// TwinCAT 3 PLC project Main
// ProgramVersion: 3.1.4022.4
// libraries:
//   Tc2_FTP, * (Beckhoff Automation GmbH)
//   Tc2_MC2, * (Beckhoff Automation GmbH)
//   Tc2_NCI, * (Beckhoff Automation GmbH)
//   Tc2_Standard, * (Beckhoff Automation GmbH)
//   Tc2_System, * (Beckhoff Automation GmbH)
//   Tc2_Utilities, * (Beckhoff Automation GmbH)
//   Tc3_IotBase, * (Beckhoff Automation GmbH)
//   Tc3_JsonXml, * (Beckhoff Automation GmbH)
//   Tc3_Module, * (Beckhoff Automation GmbH)
//   VisuSymbols,3.5.10.0,System
// project tree:
//   / GlobalTextList.TcGTLO, PlcTask.TcTTO (not stored), Visualization Manager.TcVMO (not stored)
//   GVLs/ COM.TcGVL, GVL.TcGVL
//   POUs/ commandExecute.TcPOU, ERROR.TcPOU, FTP.TcPOU, MAIN.TcPOU, POU_NCI.TcPOU, submqtt.TcPOU, commandDecoder.TcPOU
//   VISUs/ Basic.TcVIS (not stored), Visualization.TcVIS
// real-time tasks:
//   TASK PlcTask: cycle T#10ms, priority 20, ADS port 350
// motion (NC):
//   TASK NC-Task 1 SAF: cycle T#2ms, priority 4, ADS port 501
//   TASK NC-Task 1 SVB: cycle T#10ms, priority 8, ADS port 511
//   AXIS Axis X1 (id 1)
//     OtherSettings: AllowMotionCmdToSlave=true
//     encoder EncType=4
//       EncPara: ScaleFactorNumerator=40, ScaleFactorDenominator=12800, Inverse=true, MaxCount=#x0000ffff
//         SoftEndMinControl: Enable=true
//         SoftEndMaxControl: Enable=true, Range=275
//         Inc: RefSearchInverse=true, RefSyncInverse=false, RefMode=1, RefSoftSyncMask=#x0000ffff
//     drive DrvType=24
//       DrvPara: Inverse=true
//         Analog: VeloReferenz=400, ScaleFactorActTorque=0.1
//         TimeComp: TaskDelayCycles=1
//     controller CtrType=1
//       CtrPara: PriorControlFactor=1
//         PID: PosKp=25
//         Observer: BandWidth=20
//   AXIS Axis X2 (id 2)
//     OtherSettings: AllowMotionCmdToSlave=true
//     encoder EncType=4
//       EncPara: ScaleFactorNumerator=40, ScaleFactorDenominator=12800, Inverse=true, MaxCount=#x0000ffff
//         Inc: RefSoftSyncMask=#x0000ffff
//     drive DrvType=24
//       DrvPara: Inverse=true
//         Analog: VeloReferenz=400, ScaleFactorActTorque=0.1
//         TimeComp: TaskDelayCycles=1
//     controller CtrType=1
//       CtrPara: PriorControlFactor=1
//         PID: PosKp=25
//         Observer: BandWidth=20
//   AXIS Axis Y (id 4)
//     OtherSettings: AllowMotionCmdToSlave=true
//     encoder EncType=4
//       EncPara: ScaleFactorNumerator=40, ScaleFactorDenominator=12800, Inverse=true, MaxCount=#x0000ffff
//         SoftEndMinControl: Enable=true
//         SoftEndMaxControl: Enable=true, Range=275
//         Inc: RefSearchInverse=true, RefSyncInverse=false, RefMode=1, RefSoftSyncMask=#x0000ffff
//     drive DrvType=24
//       DrvPara: Inverse=true
//         Analog: VeloReferenz=400, ScaleFactorActTorque=0.1
//         TimeComp: TaskDelayCycles=1
//     controller CtrType=1
//       CtrPara: PriorControlFactor=1
//         PID: PosKp=25
//         Observer: BandWidth=20
//   AXIS Axis Z (id 3)
//     Velo: SlowManual=2, FastManual=5
//     OtherSettings: AllowMotionCmdToSlave=true
//     encoder EncType=4
//       EncPara: ScaleFactorNumerator=1, ScaleFactorDenominator=12800, MaxCount=#x0000ffff
//         Inc: RefSoftSyncMask=#x0000ffff
//     drive DrvType=24
//       Analog: VeloReferenz=10, ScaleFactorActTorque=0.1
//       TimeComp: TaskDelayCycles=1
//     controller CtrType=1
//       CtrPara: PriorControlFactor=1
//         PID: PosKp=25
//         Observer: BandWidth=20
// I/O:
//   DEVICE Device 3 (EtherCAT), AmsNetId 5.13.205.176.4.1
//     Term 1 (EK1100) [EK1100 EtherCAT Coupler (2A E-Bus)]
//       Term 2 (EL7031-0030) [EL7031-0030 1Ch. Stepper motor output stage (24V, 2.8A)]
//       Term 3 (EL7031-0030) [EL7031-0030 1Ch. Stepper motor output stage (24V, 2.8A)]
//       Term 4 (EL7031-0030) [EL7031-0030 1Ch. Stepper motor output stage (24V, 2.8A)]
//       Term 5 (EL7031-0030) [EL7031-0030 1Ch. Stepper motor output stage (24V, 2.8A)]
//       Term 6 (EL1008) [EL1008 8Ch. Dig. Input 24V, 3ms]
//       Term 7 (EL9011) [EL9011 End Terminal]
// variable links:
//   NC-Task 1 SAF/Axes/Axis X1 <-> Device 3 (EtherCAT)/Term 1 (EK1100)/Term 2 (EL7031-0030)
//     Drive/Inputs/In/nState1 @bit 3 <-> STM Status/Status/Error
//     Drive/Inputs/In/nState1 @bit 5 <-> STM Status/Status/Moving negative
//     Drive/Inputs/In/nState1 @bit 4 <-> STM Status/Status/Moving positive
//     Drive/Inputs/In/nState1 @bit 1 <-> STM Status/Status/Ready
//     Drive/Inputs/In/nState1 <-> STM Status/Status/Ready to enable
//     Drive/Inputs/In/nState1 @bit 6 <-> STM Status/Status/Torque reduced
//     Drive/Inputs/In/nState1 @bit 2 <-> STM Status/Status/Warning
//     Drive/Inputs/In/nState2 @bit 3 <-> STM Status/Status/Digital input 1
//     Drive/Inputs/In/nState2 @bit 4 <-> STM Status/Status/Digital input 2
//     Drive/Inputs/In/nState2 @bit 5 <-> STM Status/Status/Sync error
//     Drive/Inputs/In/nState2 @bit 7 <-> STM Status/Status/TxPDO Toggle
//     Drive/Inputs/In/nState4 @bit 1 <-> WcState/InputToggle
//     Drive/Inputs/In/nState4 <-> WcState/WcState
//     Drive/Outputs/Out/nCtrl1 <-> STM Control/Control/Enable
//     Drive/Outputs/Out/nCtrl1 @bit 2 <-> STM Control/Control/Reduce torque
//     Drive/Outputs/Out/nCtrl1 @bit 1 <-> STM Control/Control/Reset
//     Drive/Outputs/Out/nDataOut2[0] <-> STM Velocity/Velocity
//     Enc/Inputs/In/nDataIn1[0] <-> ENC Status compact/Counter value
//     Enc/Inputs/In/nDataIn2[0] <-> ENC Status compact/Latch value
//     Enc/Inputs/In/nState1 @bit 4 <-> ENC Status compact/Status/Counter overflow
//     Enc/Inputs/In/nState1 @bit 3 <-> ENC Status compact/Status/Counter underflow
//     Enc/Inputs/In/nState1 @bit 1 <-> ENC Status compact/Status/Latch extern valid
//     Enc/Inputs/In/nState1 @bit 2 <-> ENC Status compact/Status/Set counter done
//     Enc/Inputs/In/nState2 @bit 4 <-> ENC Status compact/Status/Status of extern latch
//     Enc/Inputs/In/nState2 @bit 5 <-> ENC Status compact/Status/Sync error
//     Enc/Inputs/In/nState2 @bit 7 <-> ENC Status compact/Status/TxPDO Toggle
//     Enc/Inputs/In/nState4 @bit 1 <-> WcState/InputToggle
//     Enc/Inputs/In/nState4 <-> WcState/WcState
//     Enc/Outputs/Out/nCtrl1 @bit 3 <-> ENC Control compact/Control/Enable latch extern on negative edge
//     Enc/Outputs/Out/nCtrl1 @bit 1 <-> ENC Control compact/Control/Enable latch extern on positive edge
//     Enc/Outputs/Out/nCtrl1 @bit 2 <-> ENC Control compact/Control/Set counter
//     Enc/Outputs/Out/nDataOut1[0] <-> ENC Control compact/Set counter value
//   NC-Task 1 SAF/Axes/Axis X2 <-> Device 3 (EtherCAT)/Term 1 (EK1100)/Term 3 (EL7031-0030)
//     Drive/Inputs/In/nState1 @bit 3 <-> STM Status/Status/Error
//     Drive/Inputs/In/nState1 @bit 5 <-> STM Status/Status/Moving negative
//     Drive/Inputs/In/nState1 @bit 4 <-> STM Status/Status/Moving positive
//     Drive/Inputs/In/nState1 @bit 1 <-> STM Status/Status/Ready
//     Drive/Inputs/In/nState1 <-> STM Status/Status/Ready to enable
//     Drive/Inputs/In/nState1 @bit 6 <-> STM Status/Status/Torque reduced
//     Drive/Inputs/In/nState1 @bit 2 <-> STM Status/Status/Warning
//     Drive/Inputs/In/nState2 @bit 3 <-> STM Status/Status/Digital input 1
//     Drive/Inputs/In/nState2 @bit 4 <-> STM Status/Status/Digital input 2
//     Drive/Inputs/In/nState2 @bit 5 <-> STM Status/Status/Sync error
//     Drive/Inputs/In/nState2 @bit 7 <-> STM Status/Status/TxPDO Toggle
//     Drive/Inputs/In/nState4 @bit 1 <-> WcState/InputToggle
//     Drive/Inputs/In/nState4 <-> WcState/WcState
//     Drive/Outputs/Out/nCtrl1 <-> STM Control/Control/Enable
//     Drive/Outputs/Out/nCtrl1 @bit 2 <-> STM Control/Control/Reduce torque
//     Drive/Outputs/Out/nCtrl1 @bit 1 <-> STM Control/Control/Reset
//     Drive/Outputs/Out/nDataOut2[0] <-> STM Velocity/Velocity
//     Enc/Inputs/In/nDataIn1[0] <-> ENC Status compact/Counter value
//     Enc/Inputs/In/nDataIn2[0] <-> ENC Status compact/Latch value
//     Enc/Inputs/In/nState1 @bit 4 <-> ENC Status compact/Status/Counter overflow
//     Enc/Inputs/In/nState1 @bit 3 <-> ENC Status compact/Status/Counter underflow
//     Enc/Inputs/In/nState1 @bit 1 <-> ENC Status compact/Status/Latch extern valid
//     Enc/Inputs/In/nState1 @bit 2 <-> ENC Status compact/Status/Set counter done
//     Enc/Inputs/In/nState2 @bit 4 <-> ENC Status compact/Status/Status of extern latch
//     Enc/Inputs/In/nState2 @bit 5 <-> ENC Status compact/Status/Sync error
//     Enc/Inputs/In/nState2 @bit 7 <-> ENC Status compact/Status/TxPDO Toggle
//     Enc/Inputs/In/nState4 @bit 1 <-> WcState/InputToggle
//     Enc/Inputs/In/nState4 <-> WcState/WcState
//     Enc/Outputs/Out/nCtrl1 @bit 3 <-> ENC Control compact/Control/Enable latch extern on negative edge
//     Enc/Outputs/Out/nCtrl1 @bit 1 <-> ENC Control compact/Control/Enable latch extern on positive edge
//     Enc/Outputs/Out/nCtrl1 @bit 2 <-> ENC Control compact/Control/Set counter
//     Enc/Outputs/Out/nDataOut1[0] <-> ENC Control compact/Set counter value
//   NC-Task 1 SAF/Axes/Axis Y <-> Device 3 (EtherCAT)/Term 1 (EK1100)/Term 5 (EL7031-0030)
//     Drive/Inputs/In/nState1 @bit 3 <-> STM Status/Status/Error
//     Drive/Inputs/In/nState1 @bit 5 <-> STM Status/Status/Moving negative
//     Drive/Inputs/In/nState1 @bit 4 <-> STM Status/Status/Moving positive
//     Drive/Inputs/In/nState1 @bit 1 <-> STM Status/Status/Ready
//     Drive/Inputs/In/nState1 <-> STM Status/Status/Ready to enable
//     Drive/Inputs/In/nState1 @bit 6 <-> STM Status/Status/Torque reduced
//     Drive/Inputs/In/nState1 @bit 2 <-> STM Status/Status/Warning
//     Drive/Inputs/In/nState2 @bit 3 <-> STM Status/Status/Digital input 1
//     Drive/Inputs/In/nState2 @bit 4 <-> STM Status/Status/Digital input 2
//     Drive/Inputs/In/nState2 @bit 5 <-> STM Status/Status/Sync error
//     Drive/Inputs/In/nState2 @bit 7 <-> STM Status/Status/TxPDO Toggle
//     Drive/Inputs/In/nState4 @bit 1 <-> WcState/InputToggle
//     Drive/Inputs/In/nState4 <-> WcState/WcState
//     Drive/Outputs/Out/nCtrl1 <-> STM Control/Control/Enable
//     Drive/Outputs/Out/nCtrl1 @bit 2 <-> STM Control/Control/Reduce torque
//     Drive/Outputs/Out/nCtrl1 @bit 1 <-> STM Control/Control/Reset
//     Drive/Outputs/Out/nDataOut2[0] <-> STM Velocity/Velocity
//     Enc/Inputs/In/nDataIn1[0] <-> ENC Status compact/Counter value
//     Enc/Inputs/In/nDataIn2[0] <-> ENC Status compact/Latch value
//     Enc/Inputs/In/nState1 @bit 4 <-> ENC Status compact/Status/Counter overflow
//     Enc/Inputs/In/nState1 @bit 3 <-> ENC Status compact/Status/Counter underflow
//     Enc/Inputs/In/nState1 @bit 1 <-> ENC Status compact/Status/Latch extern valid
//     Enc/Inputs/In/nState1 @bit 2 <-> ENC Status compact/Status/Set counter done
//     Enc/Inputs/In/nState2 @bit 4 <-> ENC Status compact/Status/Status of extern latch
//     Enc/Inputs/In/nState2 @bit 5 <-> ENC Status compact/Status/Sync error
//     Enc/Inputs/In/nState2 @bit 7 <-> ENC Status compact/Status/TxPDO Toggle
//     Enc/Inputs/In/nState4 @bit 1 <-> WcState/InputToggle
//     Enc/Inputs/In/nState4 <-> WcState/WcState
//     Enc/Outputs/Out/nCtrl1 @bit 3 <-> ENC Control compact/Control/Enable latch extern on negative edge
//     Enc/Outputs/Out/nCtrl1 @bit 1 <-> ENC Control compact/Control/Enable latch extern on positive edge
//     Enc/Outputs/Out/nCtrl1 @bit 2 <-> ENC Control compact/Control/Set counter
//     Enc/Outputs/Out/nDataOut1[0] <-> ENC Control compact/Set counter value
//   NC-Task 1 SAF/Axes/Axis Z <-> Device 3 (EtherCAT)/Term 1 (EK1100)/Term 4 (EL7031-0030)
//     Drive/Inputs/In/nState1 @bit 3 <-> STM Status/Status/Error
//     Drive/Inputs/In/nState1 @bit 5 <-> STM Status/Status/Moving negative
//     Drive/Inputs/In/nState1 @bit 4 <-> STM Status/Status/Moving positive
//     Drive/Inputs/In/nState1 @bit 1 <-> STM Status/Status/Ready
//     Drive/Inputs/In/nState1 <-> STM Status/Status/Ready to enable
//     Drive/Inputs/In/nState1 @bit 6 <-> STM Status/Status/Torque reduced
//     Drive/Inputs/In/nState1 @bit 2 <-> STM Status/Status/Warning
//     Drive/Inputs/In/nState2 @bit 3 <-> STM Status/Status/Digital input 1
//     Drive/Inputs/In/nState2 @bit 4 <-> STM Status/Status/Digital input 2
//     Drive/Inputs/In/nState2 @bit 5 <-> STM Status/Status/Sync error
//     Drive/Inputs/In/nState2 @bit 7 <-> STM Status/Status/TxPDO Toggle
//     Drive/Inputs/In/nState4 @bit 1 <-> WcState/InputToggle
//     Drive/Inputs/In/nState4 <-> WcState/WcState
//     Drive/Outputs/Out/nCtrl1 <-> STM Control/Control/Enable
//     Drive/Outputs/Out/nCtrl1 @bit 2 <-> STM Control/Control/Reduce torque
//     Drive/Outputs/Out/nCtrl1 @bit 1 <-> STM Control/Control/Reset
//     Drive/Outputs/Out/nDataOut2[0] <-> STM Velocity/Velocity
//     Enc/Inputs/In/nDataIn1[0] <-> ENC Status compact/Counter value
//     Enc/Inputs/In/nDataIn2[0] <-> ENC Status compact/Latch value
//     Enc/Inputs/In/nState1 @bit 4 <-> ENC Status compact/Status/Counter overflow
//     Enc/Inputs/In/nState1 @bit 3 <-> ENC Status compact/Status/Counter underflow
//     Enc/Inputs/In/nState1 @bit 1 <-> ENC Status compact/Status/Latch extern valid
//     Enc/Inputs/In/nState1 @bit 2 <-> ENC Status compact/Status/Set counter done
//     Enc/Inputs/In/nState2 @bit 4 <-> ENC Status compact/Status/Status of extern latch
//     Enc/Inputs/In/nState2 @bit 5 <-> ENC Status compact/Status/Sync error
//     Enc/Inputs/In/nState2 @bit 7 <-> ENC Status compact/Status/TxPDO Toggle
//     Enc/Inputs/In/nState4 @bit 1 <-> WcState/InputToggle
//     Enc/Inputs/In/nState4 <-> WcState/WcState
//     Enc/Outputs/Out/nCtrl1 @bit 3 <-> ENC Control compact/Control/Enable latch extern on negative edge
//     Enc/Outputs/Out/nCtrl1 @bit 1 <-> ENC Control compact/Control/Enable latch extern on positive edge
//     Enc/Outputs/Out/nCtrl1 @bit 2 <-> ENC Control compact/Control/Set counter
//     Enc/Outputs/Out/nDataOut1[0] <-> ENC Control compact/Set counter value
//   Main/Main Instance <-> Device 3 (EtherCAT)/Term 1 (EK1100)/Term 6 (EL1008)
//     PlcTask Inputs/GVL.bX1 <-> Channel 3/Input
//     PlcTask Inputs/GVL.bX2 <-> Channel 4/Input
//     PlcTask Inputs/GVL.bY1 <-> Channel 1/Input
//     PlcTask Inputs/GVL.bY2 <-> Channel 2/Input
//   Main/Main Instance <-> NC-Task 1 SAF/Axes/Axis X1
//     PlcTask Inputs/GVL.As_Xa.NcToPlc <-> Outputs/ToPlc
//     PlcTask Outputs/GVL.As_Xa.PlcToNc <-> Inputs/FromPlc
//   Main/Main Instance <-> NC-Task 1 SAF/Axes/Axis X2
//     PlcTask Inputs/GVL.As_Xb.NcToPlc <-> Outputs/ToPlc
//     PlcTask Outputs/GVL.As_Xb.PlcToNc <-> Inputs/FromPlc
//   Main/Main Instance <-> NC-Task 1 SAF/Axes/Axis Y
//     PlcTask Inputs/GVL.As_Y.NcToPlc <-> Outputs/ToPlc
//     PlcTask Outputs/GVL.As_Y.PlcToNc <-> Inputs/FromPlc
//   Main/Main Instance <-> NC-Task 1 SAF/Axes/Axis Z
//     PlcTask Inputs/GVL.As_Z.NcToPlc <-> Outputs/ToPlc
//     PlcTask Outputs/GVL.As_Z.PlcToNc <-> Inputs/FromPlc
//   Main/Main Instance <-> NC-Task 1 SAF/G-code
//     PlcTask Inputs/GVL.ChannelInput <-> Outputs/ToPlc
//     PlcTask Outputs/GVL.ChannelOutput <-> Inputs/FromPlc

// ---- GVLs/COM.TcGVL
{attribute 'qualified_only'}
VAR_GLOBAL
	
	bEnable		: BOOL := FALSE;
	bCouple		: BOOL := FALSE;
	bReset		: BOOL := FALSE;
	bHome		: BOOL := FALSE;

	bMoveX		: BOOL;
	bMoveY		: BOOL;
	bMoveZ		: BOOL;
		
	bSetZ		: BOOL;
	
	absX 		: INT := 0;
	absY 		: INT := 0;
	absZ 		: INT := 0;
	
	velX 		: INT := 200;	//0-400
	velY 		: INT := 200;	//0-400
	velZ 		: INT := 3;		//0-10
	
	PosX 		: LREAL;
	PosY 		: LREAL;
	PosZ 		: LREAL;
	bValid		: BOOL;
	
	bHomeDone	: BOOL;
	bHomeBusy	: BOOL;
	bMoveDone	: BOOL;
	bMoveXDone	: BOOL;
	bMoveYDone	: BOOL;
	bMoveZDone	: BOOL;
	bMoveBusy	: BOOL;
	
	bError 		: BOOL;
	
	inUSe 		: BOOL;
END_VAR

// ---- GVLs/GVL.TcGVL
{attribute 'qualified_only'}
VAR_GLOBAL
	As_Xa : AXIS_REF;
	As_Xb : AXIS_REF;
	As_Y : AXIS_REF;
	As_Z : AXIS_REF;
	
	ChannelInput AT %I* : NCTOPLC_NCICHANNEL_REF;
	ChannelOutput AT %Q* : PLCTONC_NCICHANNEL_REF;
	
	StopALL : bool;
	
	bX1 AT%I* : BOOL;
	bX2 AT%I* : BOOL;
	bY1 AT%I* : BOOL;
	bY2 AT%I* : BOOL;
	
	stReceivedData	: STRING(255);
		
END_VAR

// ---- POUs/commandExecute.TcPOU
PROGRAM commandExecute
VAR
	MCPower_Xa, MCPower_Xb, MCPower_Y, 	MCPower_Z 	: MC_Power;
	MCResetXa, MCResetXb, MCResetY, MCResetZ		: MC_Reset;

	fb_MCGearIn										: MC_GearIn;
	fb_MCGearOut									: MC_GearOut;

	fb_MCHOME_X, fb_MCHOME_Y						: MC_Home;
	fb_MoveAbs_X, fb_MoveAbs_Y, fb_MoveAbs_Z 		: MC_MoveAbsolute;
	fb_ReadX, fb_ReadY, fb_readZ 					: MC_ReadActualPosition;

	fb_SetZToZero 	: MC_SetPosition;
	
END_VAR

//Enable Axis
	MCPower_Xa(
		Axis:= GVL.As_Xa, 
		Enable:= COM.bEnable, 
		Enable_Positive:= COM.bEnable, 
		Enable_Negative:= COM.bEnable, 
		Override:= 100 );
		
	MCPower_Xb(
		Axis:= GVL.As_Xb, 
		Enable:= COM.bEnable, 
		Enable_Positive:= COM.bEnable, 
		Enable_Negative:= COM.bEnable, 
		Override:= 100 );
		
	MCPower_Y(
		Axis:= GVL.As_Y, 
		Enable:= COM.bEnable, 
		Enable_Positive:= COM.bEnable, 
		Enable_Negative:= COM.bEnable, 
		Override:= 100 );
		
	MCPower_Z(
		Axis:= GVL.As_Z, 
		Enable:= COM.bEnable, 
		Enable_Positive:= COM.bEnable, 
		Enable_Negative:= COM.bEnable, 
		Override:= 100 );

//Reset Axis
	MCResetXa(
		Axis:= GVL.As_Xa, 
		Execute:= COM.bReset );
	
	MCResetXb(
		Axis:= GVL.As_Xb, 
		Execute:= COM.bReset );

	MCResetY(
		Axis:= GVL.As_Y, 
		Execute:= COM.bReset );

	MCResetZ(
		Axis:= GVL.As_Z, 
		Execute:= COM.bReset );
	
//Couple Axis
	fb_MCGearIn(
		Master:= GVL.As_Xa, 
		Slave:= GVL.As_Xb, 
		Execute:= COM.bCouple, 
		RatioNumerator:= 1, 
		RatioDenominator:= 1 );
		
	fb_MCGearOut(
		Slave:= GVL.As_Xb,
		Execute:= NOT(COM.bCouple) );
		
//Homing
	fb_MCHOME_X(
		Axis:= GVL.As_Xa, 
		Execute:= COM.bHome AND COM.bCouple, 
		Position:= 0, 
		bCalibrationCam:= GVL.bX1 );
	
	fb_MCHOME_Y(
		Axis:= GVL.As_Y, 
		Execute:= COM.bHome AND COM.bCouple, 
		Position:= 0, 
		bCalibrationCam:= GVL.bY1 );
		
//Absolute movement
	fb_MoveAbs_X(
		Axis := GVL.As_Xa,
		Execute := COM.bMoveX AND COM.bCouple,
		Position := COM.absX,
		Velocity := COM.velX);
		
	fb_MoveAbs_Y(
		Axis := GVL.As_Y,
		Execute := COM.bMoveY,
		Position := COM.absY,
		Velocity := COM.velY);		
		
	fb_MoveAbs_Z(
		Axis := GVL.As_Z,
		Execute := COM.bMoveZ,
		Position := COM.absZ,
		Velocity := COM.velZ);		
		
//set Z postition to zero
	fb_SetZToZero(
		Axis := GVL.As_Z, 
		Execute := COM.bSetZ,
		Position := 0, 
		Mode := FALSE);

//read actual position
	fb_ReadX(Enable := TRUE, Axis := GVL.As_Xa, Position => COM.PosX);
	fb_ReadY(Enable := TRUE, Axis := GVL.As_Y, Position => COM.PosY);
	fb_ReadZ(Enable := TRUE, Axis := GVL.As_Z, Position => COM.PosZ);
	COM.bValid := fb_ReadX.Valid AND fb_ReadY.Valid AND fb_ReadZ.Valid;
	
//done = busy
	COM.bHomeBusy	:= fb_MCHOME_X.Busy OR fb_MCHOME_Y.Busy;
	COM.bMoveBusy	:= fb_MoveAbs_X.Busy OR fb_MoveAbs_Y.Busy OR fb_MoveAbs_Z.Busy;		
	
	COM.bHomeDone	:= fb_MCHOME_X.Done AND fb_MCHOME_Y.Done;
	COM.bMoveDone	:= fb_MoveAbs_X.Done AND fb_MoveAbs_Y.Done AND fb_MoveAbs_Z.Done;
	
	COM.bMoveXDone	:= fb_MoveAbs_X.Done;
	COM.bMoveYDone	:= fb_MoveAbs_Y.Done;
	COM.bMoveZDone	:= fb_MoveAbs_Z.Done;

END_PROGRAM

// ---- POUs/ERROR.TcPOU
PROGRAM ERROR
VAR
	StopX_a : MC_Stop;
	StopX_b : MC_Stop;
	StopY : MC_Stop;
	StopZ : MC_Stop;
	
	FB_AXISERRORXa, FB_AXISERRORXb, FB_AXISERRORY, FB_AXISERRORZ : MC_ReadAxisError;
	ErrorIDXa 	: DWORD;
	ErrorIDXb 	: DWORD;
	ErrorIDY 	: DWORD;
	ErrorIDZ 	: DWORD;
	ErrorAxisXa	: UDINT;
	ErrorAxisXb	: UDINT;
	ErrorAxisY	: UDINT;
	ErrorAxisZ	: UDINT;
END_VAR

// https://infosys.beckhoff.com/english.php?content=../content/1033/tccncmcplatform_fb/html/mcstop.htm&id=

//stop all
StopX_a(Axis := gvl.As_Xa,
		Execute := GVL.StopALL);

StopX_b(Axis := gvl.As_Xb,
		Execute := GVL.StopALL);

StopY(Axis := gvl.As_Y,
		Execute := GVL.StopALL);
		
StopZ(Axis := gvl.As_Z,
		Execute := GVL.StopALL);
		
FB_AxisErrorXa(Axis := gvl.As_Xa, Enable := TRUE);
FB_AxisErrorXb(Axis := gvl.As_Xb, Enable := TRUE);
FB_AxisErrorY(Axis := gvl.As_Y, Enable := TRUE);
FB_AxisErrorZ(Axis := gvl.As_Z, Enable := TRUE);

ErrorIDXa 	:= FB_AxisErrorXa.ErrorID;
ErrorIDXb 	:= FB_AxisErrorXb.ErrorID;
ErrorIDY 	:= FB_AxisErrorY.ErrorID;
ErrorIDZ 	:= FB_AxisErrorZ.ErrorID;

ErrorAxisXa	:= FB_AxisErrorXa.AxisErrorID;
ErrorAxisXb	:= FB_AxisErrorXb.AxisErrorID;
ErrorAxisY	:= FB_AxisErrorY.AxisErrorID;
ErrorAxisZ	:= FB_AxisErrorZ.AxisErrorID;

END_PROGRAM

// ---- POUs/FTP.TcPOU
PROGRAM FTP
VAR
 		RisingEdge              : R_TRIG;
        startstop               : BOOL;

        state                   : BYTE;

        FB_FTP_Open1            : FB_FTP_Open;
        FB_FTP_FileList1                : FB_FTP_FileList;
        FB_FTP_Close1           : FB_FTP_Close;

        busy                    : BOOL;
        err                     : BOOL;
        errid                   : UDINT;

        handle                  : T_HFTP;
        
        FileList                        : ARRAY [0..MAX_FILELIST_ITEMS] OF STRING;
        Items                   : UDINT;       
END_VAR

//https://download.beckhoff.com/download/document/automation/twincat3/TF6300_TC3_FTP_CLIENT_EN.pdf

//ftp://<CX1000 IP Address>

//testing
RisingEdge(CLK:= startstop);
IF RisingEdge.Q THEN
        state := 1;
END_IF

CASE state OF
        0:
                ;

        1:
                FB_FTP_Open1(
                        sNetID:= '5.0.252.142.1.1',
                        sHost:= '172.16.9.223',
                        nPort:= 21,
                        sUsername:= 'TestUser',
                        sPassword:= 'TestPwd123',
                        bExecute:= TRUE,
                        tTimeout:= T#15s,
                        bBusy=> busy,
                        bError=> err,
                        nErrId=> errid,
                        hFTP=> handle);

                IF NOT busy AND NOT err THEN
                        FB_FTP_Open1(bExecute:= FALSE);
                        state := 2;
                END_IF

        2:
                FB_FTP_FileList1(
                        sNetID:= '5.0.252.142.1.1',
                        hFTP:= handle,
                        sMask:= '*.txt',
                        nIndex:= 0,
                        pList:= ADR(FileList),
                        cbList:= SIZEOF(FileList),
                        bExecute:= TRUE,
                        tTimeout:= T#15s,
                        bBusy=> busy,
                        bError=> err,
                        nErrID=> errid,
                        nItems=> Items);

                IF NOT busy AND NOT err THEN
                        FB_FTP_FileList1(bExecute:= FALSE);
                        state := 3;
                END_IF

        3:
                FB_FTP_Close1(
                        sNetID:= '5.0.252.142.1.1',
                        hFTP:= handle,
                        bExecute:= TRUE,
                        tTimeout:= T#15s,
                        bBusy => busy,
                        bError => err,
                        nErrId => errid);

                IF NOT busy AND NOT err THEN
                        FB_FTP_Close1(bExecute:= FALSE);
                        state := 0;
                END_IF

END_CASE

END_PROGRAM

// ---- POUs/MAIN.TcPOU
PROGRAM MAIN
VAR
	
END_VAR

//main program
	//POU_NCI();

//SUBMQTT Connection and receiving
	//submqtt();

//FTP
	//FTP();

//AT Commands
	commandDecoder();
	commandExecute();

//Error
	ERROR();

END_PROGRAM

// ---- POUs/commandDecoder.TcPOU
PROGRAM commandDecoder
VAR
	command 	: STRING(255);
	Head_Loaded : STRING;
	index 		: INT := 0;
	
	actualX 	: LREAL;
	actualY 	: LREAL;
	actualZ 	: Lreal;
	
	wait100ms : TON;
	
END_VAR

command := GVL.stReceivedData;
command := F_ToLCase(command);
GVL.stReceivedData := '';

wait100ms(IN := COM.bEnable, pt := T#500MS);

CASE index OF
	0:	//commands
		COM.bEnable := FALSE;
		COM.bCouple := FALSE;
		COM.bHome 	:= FALSE;
		COM.inUSe 	:= FALSE;
		
		IF 		(command = 'reset') THEN
			index := 10;
			command := '';
    	ELSIF 	(command = 'homing') THEN
			index := 100;
			command := '';
		ELSIF 	(command = 'z to zero') THEN
			index := 110;
			command := '';
		ELSIF 	(command = 'set vel') THEN
			index := 120;
			command := '';
		ELSIF 	(command = 'go xyz') THEN
			index := 200;
			command := '';
		ELSIF 	(command = 'go x') THEN
			index := 210;
			command := '';
		ELSIF 	(command = 'go y') THEN
			index := 220;
			command := '';
		ELSIF 	(command = 'go z') THEN
			index := 230;
			command := '';
		ELSIF 	(command = 'exec gcode') THEN
			index := 250;
			command := '';
		ELSIF 	(command = 'read pos') THEN
			index := 300;
			command := '';
		ELSIF 	(command = 'error') THEN
			index := 999;
			command := '';
		ELSE
			index := 0;
		END_IF;
		
	10: //reset
		COM.bReset 	:= TRUE;
		COM.bReset 	:= FALSE;
		
		COM.bEnable := FALSE;
		COM.bCouple := FALSE;
		COM.bHome 	:= FALSE;
		COM.inUSe 	:= FALSE;
		COM.bMoveX 	:= FALSE;
		COM.bMoveY 	:= FALSE;
		COM.bMoveZ 	:= FALSE;
		
		index 		:= 0;
		
	100: //Homing
		COM.bEnable := TRUE;
		COM.bCouple := TRUE;
		COM.bHome 	:= TRUE;
		
		IF COM.bHomeBusy THEN
			COM.inUSe 	:= TRUE;
		ELSE
			COM.inUSe 	:= FALSE;
		END_IF
		
		IF COM.bHomeDone THEN
			COM.bEnable := FALSE;
			COM.bCouple := FALSE;
			COM.bHome 	:= FALSE;
			COM.inUSe 	:= FALSE;
			index 	:= 0;
		END_IF
		
	110: //set Z position to zero
			COM.bSetZ 		:= TRUE;
			IF (COM.PosZ = 0 AND COM.bValid) THEN
				COM.bSetZ 	:= FALSE;
				index 		:= 0;
			END_IF
			
	120: //Set velocity
		COM.velX := 200;
		COM.velY := 200;
		COM.velZ := 2;
		index 		:= 0;
	
	200: //Go to xyz Pos
    	COM.absX := 100;
		COM.absY := 100;
		COM.absZ := 0;
		
		COM.bEnable := TRUE;
		COM.bCouple := TRUE;
		
		IF wait100ms.Q THEN 
			COM.bMoveX 	:= TRUE;
			COM.bMoveY 	:= TRUE;
			COM.bMoveZ 	:= TRUE;
		END_IF
		
		IF COM.bHomeBusy THEN
			COM.inUSe 	:= TRUE;
		ELSE
			COM.inUSe 	:= FALSE;
		END_IF
		
		IF COM.bMoveDone THEN
			COM.bEnable := FALSE;
			COM.bCouple := FALSE;
			COM.inUSe 	:= FALSE;
			COM.bMoveX 	:= FALSE;
			COM.bMoveY 	:= FALSE;
			COM.bMoveZ 	:= FALSE;
			index 	:= 0;
		END_IF
		
	210: //Go X Pos
	    COM.absX := 50;
		COM.bEnable := TRUE;
		COM.bCouple := TRUE;
		
		IF wait100ms.Q THEN 
			COM.bMoveX 	:= TRUE;
		END_IF
		
		IF COM.bHomeBusy THEN
			COM.inUSe 	:= TRUE;
		ELSE
			COM.inUSe 	:= FALSE;
		END_IF
		
		IF COM.bMoveXDone THEN
			COM.bEnable := FALSE;
			COM.bCouple := FALSE;
			COM.inUSe 	:= FALSE;
			COM.bMoveX 	:= FALSE;
			index 	:= 0;
		END_IF

	220: //Go Y Pos
		COM.bEnable := TRUE;
		COM.absY := 50;
		
		IF wait100ms.Q THEN 
			COM.bMoveY 	:= TRUE;
		END_IF
				
		IF COM.bHomeBusy THEN
			COM.inUSe 	:= TRUE;
		ELSE
			COM.inUSe 	:= FALSE;
		END_IF
		
		IF COM.bMoveYDone THEN
			COM.bEnable := FALSE;
			COM.bCouple := FALSE;
			COM.inUSe 	:= FALSE;
			COM.bMoveY 	:= FALSE;
			index 	:= 0;
		END_IF

	230: //Go Z Pos
		COM.absZ := -1;
		COM.bEnable := TRUE;
		
		IF wait100ms.Q THEN 
			COM.bMoveZ 	:= TRUE;
		END_IF
		
		IF COM.bHomeBusy THEN
			COM.inUSe 	:= TRUE;
		ELSE
			COM.inUSe 	:= FALSE;
		END_IF
		
		IF COM.bMoveZDone THEN
			COM.bEnable := FALSE;
			COM.bCouple := FALSE;
			COM.inUSe 	:= FALSE;
			COM.bMoveZ 	:= FALSE;
			index 	:= 0;
		END_IF
		
	250: //Execute Gcode--------------------------------------------------------------------------------------------
		
	300: //Read XYZ
		actualX 	:= COM.PosX;
		actualY 	:= COM.Posy;
		actualZ 	:= COM.PosZ;
		IF COM.bValid THEN
			index 	:= 0;
		END_IF

	999: //error
			COM.bEnable := FALSE;
			IF(command = 'reset')THEN
				index := 0;
			END_IF

	ELSE //errorstate
	index := 0;
END_CASE;

END_PROGRAM

// ---- POUs/POU_NCI.TcPOU
PROGRAM POU_NCI
VAR
	
	fb_BuildGroup: CfgBuild3DGroup;
	fb_ReconfigGroup: CfgReconfigGroup;
	fb_LoadProg: ItpLoadProgEx;
	fb_StartStop: ItpStartStopEx;
	fb_Reset: ItpResetEx2;
	
	bBuildGroup: BOOL;
	bLoad: BOOL;
	bStart: BOOL;
	bStop: BOOL;
	bReset: BOOL;
	
END_VAR

fb_BuildGroup(
	bExecute:= bBuildGroup, 
	nGroupId:= GVL.ChannelInput.GrpId, 
	nXAxisId:= GVL.As_Xa.NcToPlc.AxisId, 
	nYAxisId:= GVL.As_Y.NcToPlc.AxisId, 
	nZAxisId:= GVL.As_Z.NcToPlc.AxisId, 
	tTimeOut:= T#1S );
	
fb_ReconfigGroup(
	bExecute:= NOT(bBuildGroup), 
	nGroupId:= GVL.ChannelInput.GrpId, 
	tTimeOut:= T#1S );
	
ItpSetOverridePercent(fOverridePercent:= 100, sPlcToNci:= GVL.ChannelOutput);

fb_LoadProg(
	sNciToPlc:= GVL.ChannelInput, 
	bExecute:= bLoad, 
	sPrg:= '\HARD DISK\TWINCAT\Mc\Nci\Gcode_test1.nc', 
	nLength:= LEN('\HARD DISK\TWINCAT\Mc\Nci\Gcode_test1.nc'), 
	tTimeOut:= T#1S );
	
fb_StartStop(
	bStart:= bStart, 
	bStop:= bStop, 
	tTimeOut:= T#1S, 
	sNciToPlc:= GVL.ChannelInput );
	
fb_Reset(
	bExecute:= bReset, 
	tTimeOut:= T#1S, 
	sNciToPlc:= GVL.ChannelInput );

END_PROGRAM

// ---- POUs/submqtt.TcPOU
PROGRAM submqtt
VAR
	fbMqttClient : FB_IotMqttClient;
	bSetParameter : BOOL := TRUE;
	bConnect : BOOL := TRUE;
	
	(* received message *)
	bSubscribed : BOOL;
	sTopicSub : STRING(255) := 'hermes/intent/#';//GeneraalAlfa:machineState
	{attribute 'TcEncoding':='UTF-8'}
	sTopicRcv : STRING(255);
	{attribute 'TcEncoding':='UTF-8'}
	sPayloadRcv : STRING(2047);
	fbMessageQueue : FB_IotMqttMessageQueue;
	fbMessage : FB_IotMqttMessage;
	
	hrErrorOccurred : HRESULT; // contains the latest occurred error
	
	(* JSON *)
	fbJson 			: FB_JsonDomParser;
	jsonDoc 		: SJsonValue;
	jsonProp		: SJsonValue;
	jsonValue		: SJsonValue;
	bHasMember		: BOOL;
END_VAR

IF bSetParameter THEN
	bSetParameter := FALSE;
	fbMqttClient.sHostName:= '169.254.239.248';
	fbMqttClient.nHostPort:= 1883;
//	fbMqttClient.sClientId:= 'POZ_PLC'; 
	fbMqttClient.sTopicPrefix:= ''; 
//	fbMqttClient.nKeepAlive:= 60; 
//	fbMqttClient.sUserName:= ;
//	fbMqttClient.sUserPassword:= ; 
//	fbMqttClient.stWill:= ; 
//	fbMqttClient.stTLS:= ;
	fbMqttClient.ipMessageQueue := fbMessageQueue;
END_IF

fbMqttClient.Execute(bConnect);
IF fbMqttClient.bError THEN
	// add your error logging here
	hrErrorOccurred := fbMqttClient.hrErrorCode;
END_IF

IF fbMessageQueue.nQueuedMessages > 0 THEN
	IF fbMessageQueue.Dequeue(fbMessage:=fbMessage) THEN
		fbMessage.GetTopic(pTopic:=ADR(sTopicRcv), nTopicSize:=SIZEOF(sTopicRcv) );
		fbMessage.GetPayload(pPayload:=ADR(sPayloadRcv), nPayloadSize:=SIZEOF(sPayloadRcv), bSetNullTermination:=FALSE);
	END_IF
END_IF

IF fbMqttClient.bConnected THEN
	IF NOT bSubscribed THEN
		bSubscribed := fbMqttClient.Subscribe(sTopic:=sTopicSub, eQoS:=TcIotMqttQos.AtMostOnceDelivery);
		IF fbMqttClient.bError THEN
			// add your error logging here
			hrErrorOccurred := fbMqttClient.hrErrorCode;
		END_IF
	END_IF
END_IF

(* Retrieve JSON content *)
jsonDoc := fbJson.ParseDocument(sPayloadRcv);
bHasMember := fbJson.HasMember(jsonDoc, 'input');
IF (bHasMember) THEN
	  bHasMember := FALSE;
	  jsonProp := fbJson.FindMember(jsonDoc, 'input');
	  GVL.stReceivedData := fbJson.GetString(jsonProp);
END_IF

END_PROGRAM

// ---- GlobalTextList.TcGTLO
TEXTLIST GlobalTextList
  943 = 'Absolute'
  163 = 'Couple'
  730 = 'Group'
  610 = 'Home'
  23 = 'Load'
  172 = 'move abs X'
  424 = 'Move abs X'
  68 = 'move abs Y'
  700 = 'Move abs Y'
  459 = 'move ABS z'
  52 = 'move abs z'
  760 = 'move abs Z'
  258 = 'Move abs Z'
  193 = 'move rel X'
  135 = 'Move rel X'
  829 = 'move rel Y'
  787 = 'Move rel Y'
  698 = 'move rel z'
  917 = 'move rel Z'
  750 = 'Move rel z'
  793 = 'Niet gebruiken'
  769 = 'Reconfig'
  653 = 'Relative'
  187 = 'Reset'
  285 = 'set z on pos 0'
  244 = 'Set Z pos to 0'
  127 = 'Start'
  887 = 'Stop'
  966 = 'STOP'
END_TEXTLIST

// ---- VISUs/Visualization.TcVIS
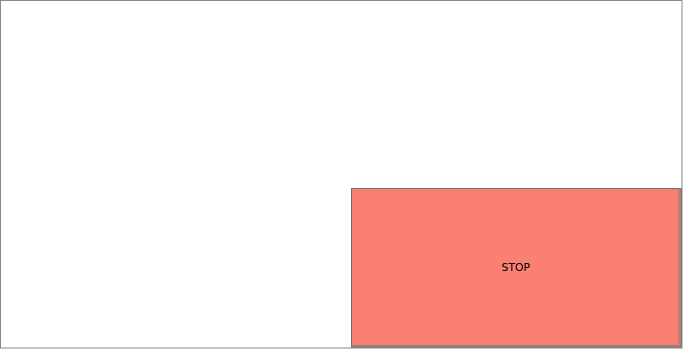
VISUALIZATION Visualization  // 683x349
    Button (351,188 330x159), "STOP", colour toggle: GVL.StopALL
        toggle GVL.StopALL
END_VISUALIZATION
